// TIA Portal V19 export
VAR_GLOBAL   // PLC tag table "00_A02_MB2_Tower"
   A02_Segnalazione_Scarico_Dopo_Taglio_Bu_SL202 AT %Q122.4 : Bool;   // 371HL3
   A02_TowerHorn_SL201 AT %Q122.3 : Bool;   // 371HA1
   A02_TowerLampYellow_SL201 AT %Q122.1 : Bool;   // 371HL1
   A02_TowerLampWhite_SL201 AT %Q122.2 : Bool;   // 371HL2
   MB2_Pb_Reset_Anomalie AT %I110.6 : Bool;   // 305SH1
   MB2_Pb_Start_Ciclo_Area03 AT %I110.7 : Bool;   // 305SH2
   MB2_Pb_Stop_Ciclo_Area03 AT %I111.0 : Bool;   // 305SB1
   MB2_Pb_Manuale_Area02 AT %I111.1 : Bool;   // 305SA1
   MB2_Pb_Automatico_Area02 AT %I111.2 : Bool;   // 305SA1
   MB2_Pb_Start_Ciclo_Area02 AT %I111.3 : Bool;   // 305SH3
   MB2_Pb_Stop_Ciclo_Area02 AT %I111.4 : Bool;   // 305SB2
   MB2_Pb_Start_Ciclo_Area01 AT %I111.5 : Bool;   // 306SH1
   MB2_Pb_Stop_Ciclo_Area01 AT %I111.6 : Bool;   // 306SB1
   MB2_Pb_Avanti_Pezzo AT %I111.7 : Bool;   // 306SB2
   MB2_Pb_Comando_Manuale_Jog_Plus AT %I112.0 : Bool;   // 306SA1
   MB2_Pb_Comando_Manuale_Jog_Menus AT %I112.1 : Bool;   // 306SA1
   MB2_Pb_Materiale_Fwd AT %I112.2 : Bool;   // 306SA2
   MB2_Pb_Materiale_Bwd AT %I112.3 : Bool;   // 306SA2
   MB2_Pb_LIBERO AT %I112.6 : Bool;   // 307 - LIBERO
   MB2_Lp_Reset_Anomalie AT %Q110.6 : Bool;   // 305SH1
   MB2_Lp_Start_Ciclo_Area03 AT %Q110.7 : Bool;   // 305SH2
   MB2_Lp_Abilitazione_Automatico_Area02 AT %Q111.0 : Bool;   // 305HL1
   MB2_Lp_Start_Ciclo_Area02 AT %Q111.1 : Bool;   // 305SH3
   MB2_Lp_Start_Ciclo_Area01 AT %Q111.2 : Bool;   // 306SH1
   MB2_Lp_Comando_Manuale_Jog_Plus AT %Q111.3 : Bool;   // 306SA1
   MB2_Lp_LIBERO AT %Q111.5 : Bool;   // 307 - LIBERO
   MB2_Pb_Carriage_Zero AT %I112.4 : Bool;
   MB2_Lp_Carriage_Zero AT %Q111.4 : Bool;   // 306SA1
END_VAR
